TYPE "MES_Err"
VERSION : 0.1
// Block: MES_Err
   STRUCT
      Presence : Bool;
      Code : DInt;
      Description : String;
   END_STRUCT;

END_TYPE
